{attribute 'qualified_only'}
{attribute 'strict'}
TYPE EDataType :
(
	none := 0,
	dont_care := 1,
	binary := 2,
	numeric := 3,
	string_t := 4
);
END_TYPE

(* stored: Version 1.1.0.1, ProductVersion 3.1.4024.9
   DUT EDataType: Id {dff9ff80-267d-44cb-ac55-ea501dcc703e} *)
